TYPE DUT_Control_Base :
STRUCT
	Open :BOOL;
	Close :BOOL;
	Reset :BOOL;
	Interlock :BOOL;
	Simulation :BOOL;
END_STRUCT
END_TYPE

(* stored: Version 1.1.0.1, ProductVersion 3.1.4024.12
   DUT DUT_Control_Base: Id {b6e1d523-0f0a-41db-aa44-7681e860b370} *)
